{attribute 'linkalways'} 
{attribute 'no_explicit_call' := 'This FB is a CLASS and must be accessed using methods or properties'}
{attribute 'enable_dynamic_creation'}
FUNCTION_BLOCK GetBlueprintsRpcHandler IMPLEMENTS I_AsynchronousRpcHandler
VAR
	nodeFactory : I_NodeFactory;
END_VAR

METHOD Handle
VAR_INPUT
	Parameters : I_Deserializer;
	Response : I_AsynchronousRpcResponse;
END_VAR
VAR
	getBlueprintsVisitor : GetBlueprintsVisitor;
	getPaginatedBlueprintsVisitor : GetPaginatedBlueprintsVisitor;
	visitor : I_NodeFactoryVisitor;
	serializer : I_Serializer;
	feedback : DeserializerFeedback;
	offset : UDINT;
	maxLimit : UDINT;
END_VAR
IF nodeFactory = 0 THEN
	Response.RejectWithMessage('GetBlueprintsRpcHandler has not been initialized with a valid nodeFactory object');
	RETURN;
END_IF

serializer := Response.GetSerializer();

IF Parameters.TryGetKeyUdint('offset', offset, feedback) AND_THEN Parameters.TryGetKeyUdint('limit', maxLimit, feedback) THEN
	// if the offset and limit are provide then use the paginated visitor
	getPaginatedBlueprintsVisitor.Initialize(serializer, offset, maxlimit);
	visitor := getPaginatedBlueprintsVisitor;
ELSE
	// if the offset and limit are not supplied then try to get all blueprints
	getBlueprintsVisitor.Initialize(serializer);
	visitor := getPaginatedBlueprintsVisitor;
END_IF

nodeFactory.Accept(visitor);
Response.CompleteWithSerializer(serializer);
serializer.Dispose();
END_METHOD

METHOD PUBLIC Initialize
VAR_INPUT
	NodeFactory : I_NodeFactory;
END_VAR
THIS^.nodeFactory := NodeFactory;
END_METHOD

END_FUNCTION_BLOCK

(* stored: Version 1.1.0.1, ProductVersion 3.1.4024.13
   POU GetBlueprintsRpcHandler: Id {c8f66f90-e7e3-49d6-b7b6-2f16dc6e40e9}, SpecialFunc None
   Method Handle: Id {b0d553f5-6d18-4f5a-ac74-32ac309a6ede}
   Method Initialize: Id {0d327fe8-8e2a-41ef-ac2a-53373485afd6} *)
